TYPE "PL_Dig"
VERSION : 0.1
   STRUCT
      Value : Bool;
      ST : Byte := 16#80;
   END_STRUCT;

END_TYPE

